// TIA Portal project "array_tanimlama" (V18)

(* hardware
DEVICE "S7-1200 station_1"  S7-1200 Station
   slot 0: "Rack_0"  S7-1200 Rack  Rack  V1.0
   slot 1: "PLC_1"  CPU 1214C AC/DC/Rly  6ES7 214-1BG40-0XB0  V4.6
*)

// ===== PLC "PLC_1"  CPU 1214C AC/DC/Rly =====

VAR_GLOBAL   // PLC tag table "Default tag table"
   "Tag_1" AT %Q0.2 : Bool;
   "Tag_2" AT %MW4 : Int;
END_VAR

DATA_BLOCK "Data_block_1"   // DB1
{ S7_Optimized_Access := 'TRUE' }
VERSION : 0.1
   VAR
      SICAKLIKLAR : Array[0..10] of Int;
   END_VAR
BEGIN
   SICAKLIKLAR[0] := 10;
   SICAKLIKLAR[1] := 20;
   SICAKLIKLAR[2] := 30;
   SICAKLIKLAR[3] := 40;
   SICAKLIKLAR[4] := 50;
   SICAKLIKLAR[5] := 60;
   SICAKLIKLAR[6] := 70;
   SICAKLIKLAR[7] := 80;
   SICAKLIKLAR[8] := 90;
   SICAKLIKLAR[9] := 100;
   SICAKLIKLAR[10] := 110;
END_DATA_BLOCK

DATA_BLOCK "Data_block_2"   // DB2
{ S7_Optimized_Access := 'TRUE' }
VERSION : 0.1
   VAR
      BASINÇ : Array[0..5, 0..4] of Int;
   END_VAR
BEGIN
   BASINÇ[0,0] := 10;
   BASINÇ[0,1] := 20;
   BASINÇ[0,2] := 30;
   BASINÇ[0,3] := 40;
   BASINÇ[0,4] := 50;
   BASINÇ[1,0] := 60;
   BASINÇ[1,1] := 70;
   BASINÇ[1,2] := 80;
   BASINÇ[1,3] := 90;
   BASINÇ[1,4] := 100;
   BASINÇ[2,0] := 110;
   BASINÇ[2,1] := 115;
   BASINÇ[2,2] := 120;
   BASINÇ[2,3] := 125;
   BASINÇ[2,4] := 130;
   BASINÇ[3,0] := 140;
   BASINÇ[3,1] := 155;
   BASINÇ[3,2] := 160;
   BASINÇ[3,3] := 200;
   BASINÇ[3,4] := 221;
   BASINÇ[4,0] := 225;
   BASINÇ[4,1] := 230;
   BASINÇ[4,2] := 2450;
   BASINÇ[4,3] := 250;
   BASINÇ[4,4] := 255;
   BASINÇ[5,0] := 256;
   BASINÇ[5,1] := 260;
   BASINÇ[5,2] := 265;
   BASINÇ[5,3] := 268;
   BASINÇ[5,4] := 180;
END_DATA_BLOCK

DATA_BLOCK "Data_block_3"   // DB3
{ S7_Optimized_Access := 'TRUE' }
VERSION : 0.1
   VAR
      OKUNAN_dEGER : Array[0..6, 9..17, 0..5] of Int;
   END_VAR
BEGIN
END_DATA_BLOCK

ORGANIZATION_BLOCK "Main"   // OB1, LAD, ProgramCycle
TITLE = "Main Program Sweep (Cycle)"
{ S7_Optimized_Access := 'TRUE' }
VERSION : 0.1
   VAR_INPUT
      Initial_Call : Bool;   // Initial call of this OB
      Remanence : Bool;   // =True, if remanent data are available
   END_VAR
BEGIN

REGION Network 1
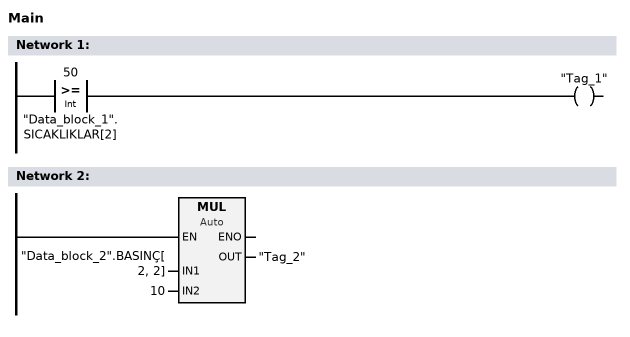
   RUNG wire#powerrail
      { S7_Templates := "SrcType := Int" } GE_Contact(in1 := 50, in2 := "Data_block_1".SICAKLIKLAR[2])
      Coil( "Tag_1" )
   END_RUNG
   // the same network as SCL:
   "Tag_1" := 50 >= "Data_block_1".SICAKLIKLAR[2];
END_REGION

REGION Network 2
   RUNG wire#powerrail
      Mul(in1 := "Data_block_2".BASINÇ[2, 2], in2 := 10, out => "Tag_2")
   END_RUNG
   // the same network as SCL:
   "Tag_2" := "Data_block_2".BASINÇ[2, 2] * 10;
END_REGION
END_ORGANIZATION_BLOCK